// TwinCAT 3 PLC project Study0725
// ProgramVersion: 3.1.4023.0
// libraries:
//   Tc2_Standard, * (Beckhoff Automation GmbH)
//   Tc2_System, * (Beckhoff Automation GmbH)
//   Tc3_Module, * (Beckhoff Automation GmbH)
// project tree:
//   / PlcTask.TcTTO
//   POUs/ MAIN.TcPOU
// real-time tasks:
//   TASK PlcTask: cycle T#10ms, priority 20, ADS port 350
//   TASK PlcTask1: cycle T#10ms, priority 21, ADS port 351

CONFIGURATION Study0725
    RESOURCE PLC ON TwinCAT3
        TASK PlcTask(INTERVAL := T#10ms, PRIORITY := 21);
        PROGRAM MAIN WITH PlcTask : MAIN;
    END_RESOURCE
END_CONFIGURATION

// ---- POUs/MAIN.TcPOU
PROGRAM MAIN
VAR
	BOOL1 AT %MX0.0:BOOL;
	ib: INT;
	Tool1: TON;
	stat: BOOL;
	tt: BOOL;
	ss: BOOL;
	CTU1:CTU;
END_VAR

ib:=1;
Tool1(IN:= ss, PT:=t#3s , Q=> , ET=> );
CTU1(
	CU:= , 
	RESET:= , 
	PV:= , 
	Q=> , 
	CV=> );

END_PROGRAM
